FUNCTION_BLOCK IOSelector (* Basic Function Block Type *)
  (* Standard: 61499-2 *)
  (* Version 0.0, 11/23/2016, chivdan, nxtControl GmbH, Template *)
  PACKAGE Main;
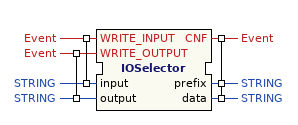
  EVENT_INPUT
    WRITE_INPUT WITH input; (* Normal Execution Request *)
    WRITE_OUTPUT WITH output;
  END_EVENT
  EVENT_OUTPUT
    CNF WITH prefix, data; (* Execution Confirmation *)
  END_EVENT
  VAR_INPUT
    input : STRING; (* Input event qualifier *)
    output : STRING;
  END_VAR
  VAR_OUTPUT
    prefix : STRING;
    data : STRING; (* Output event qualifier *)
  END_VAR
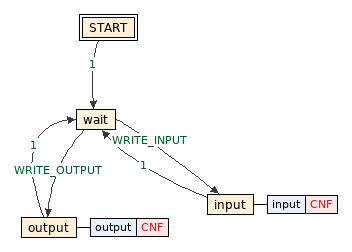
  EC_STATES
    START; (* Initial State *)
    wait; (* Normal execution *)
    input : input -> CNF;
    output : output -> CNF;
  END_STATES
  EC_TRANSITIONS
    START TO wait := 1;
    wait TO input := WRITE_INPUT;
    wait TO output := WRITE_OUTPUT;
    input TO wait := 1;
    output TO wait := 1;
  END_TRANSITIONS
  ALGORITHM INIT IN ST: (* Initialization algorithm *)
;
  END_ALGORITHM
  ALGORITHM output IN ST: (* Normally executed algorithm *)
;
prefix:='out=CNF[';
data:=output;
  END_ALGORITHM
  ALGORITHM input IN ST:
prefix:='in=REQ[';
data:=input;
  END_ALGORITHM
END_FUNCTION_BLOCK
